// TIA Portal V19 export
DATA_BLOCK "HMI"   // DB86
{ S7_Optimized_Access := 'TRUE' }
// stored: MemoryReserve 100
   VAR
      HOOTER_RESET : Bool;
      M1_SUGAR : Bool;
      M1_MFG : Bool;
      M1_STORAGE_1 : Bool;
      M1_STORAGE_2 : Bool;
      M1_MIXING : Bool;
      M2_MFG : Bool;
      M2_STORAGE_1 : Bool;
      M2_STORAGE_2 : Bool;
      M2_MIXING : Bool;
   END_VAR
BEGIN
END_DATA_BLOCK
